// ---- DUTs/IO/Topology/Beckhoff_EK12xxEK1122_F8B8118B.TcDUT
{attribute 'GeneratedUsingTerminal: EK1122-0000-0018'}
{attribute addProperty BoxType "EK1122-0000-0018"}
{attribute addProperty Id "Beckhoff_EK12xxsub_EK1100EK1100_1FC0878B2A_0002_EK1200_7000_0000EK1200_013D0B490A_0001_EK1200_5000_0000EK1200_013D0B490"}
{attribute addProperty CRC "4172812683"}
{attribute addProperty Size "2"}
{attribute addProperty Name "Beckhoff EK12xxEK1122"}
TYPE Beckhoff_EK12xxEK1122_F8B8118B EXTENDS EK1122_1FC0878B :
STRUCT
	{attribute addProperty Name "Beckhoff EK12xxsub EK1100"}
	{attribute addProperty PreviousPort "Beckhoff EK12xxEK1122 : D"}
	Beckhoff_EK12xxsub_EK1100 : EK1100_1FC0878B;
	{attribute addProperty Name "A_0002(EK1200-7000-0000)"}
	{attribute addProperty PreviousPort "Beckhoff EK12xxsub EK1100 : C"}
	A_0002_EK1200_7000_0000 : EK1200_013D0B49;
	{attribute addProperty Name "A_0001(EK1200-5000-0000)"}
	{attribute addProperty PreviousPort "Beckhoff EK12xxsub EK1100 : C"}
	A_0001_EK1200_5000_0000 : EK1200_013D0B49;
END_STRUCT
END_TYPE

// ---- DUTs/IO/Topology/Beckhoff_EK12xx_F07DE953.TcDUT
{attribute 'GeneratedUsingTerminal: EK1100-0000-0018'}
{attribute addProperty BoxType "EK1100-0000-0018"}
{attribute addProperty Id "Beckhoff_EK12xxEK1122Beckhoff_EK12xxEK1122_F8B8118B2"}
{attribute addProperty CRC "4034783571"}
{attribute addProperty Size "2"}
{attribute addProperty Name "Beckhoff EK12xx"}
TYPE Beckhoff_EK12xx_F07DE953 EXTENDS EK1100_1FC0878B :
STRUCT
	{attribute addProperty Name "Beckhoff EK12xxEK1122"}
	{attribute addProperty PreviousPort "Beckhoff EK12xx : B"}
	Beckhoff_EK12xxEK1122 : Beckhoff_EK12xxEK1122_F8B8118B;
END_STRUCT
END_TYPE

// ---- DUTs/IO/Topology/Beckhoff_EK13xxEK1122_30D1B042.TcDUT
{attribute 'GeneratedUsingTerminal: EK1122-0000-0018'}
{attribute addProperty BoxType "EK1122-0000-0018"}
{attribute addProperty Id "Beckhoff_EK13xxsub_EK1100EK1100_1FC0878B2A_0001_EK1300_0000_0017EK1300_6BC01D146"}
{attribute addProperty CRC "819048514"}
{attribute addProperty Size "8"}
{attribute addProperty Name "Beckhoff EK13xxEK1122"}
TYPE Beckhoff_EK13xxEK1122_30D1B042 EXTENDS EK1122_1FC0878B :
STRUCT
	{attribute addProperty Name "Beckhoff EK13xxsub EK1100"}
	{attribute addProperty PreviousPort "Beckhoff EK13xxEK1122 : D"}
	Beckhoff_EK13xxsub_EK1100 : EK1100_1FC0878B;
	{attribute addProperty Name "A_0001(EK1300-0000-0017)"}
	{attribute addProperty PreviousPort "Beckhoff EK13xxsub EK1100 : C"}
	A_0001_EK1300_0000_0017 : EK1300_6BC01D14;
END_STRUCT
END_TYPE

// ---- DUTs/IO/Topology/Beckhoff_EK13xx_7663BCA8.TcDUT
{attribute 'GeneratedUsingTerminal: EK1100-0000-0018'}
{attribute addProperty BoxType "EK1100-0000-0018"}
{attribute addProperty Id "Beckhoff_EK13xxEK1122Beckhoff_EK13xxEK1122_30D1B0428A_0003_EK1322_0000_0017EK1322_6BC01D146A_0002_EK1310_0000_0017EK1310_6BC01D146"}
{attribute addProperty CRC "1986247848"}
{attribute addProperty Size "20"}
{attribute addProperty Name "Beckhoff EK13xx"}
TYPE Beckhoff_EK13xx_7663BCA8 EXTENDS EK1100_1FC0878B :
STRUCT
	{attribute addProperty Name "Beckhoff EK13xxEK1122"}
	{attribute addProperty PreviousPort "Beckhoff EK13xx : B"}
	Beckhoff_EK13xxEK1122 : Beckhoff_EK13xxEK1122_30D1B042;
	{attribute addProperty Name "A_0003(EK1322-0000-0017)"}
	{attribute addProperty PreviousPort "Beckhoff EK13xxEK1122 : C"}
	A_0003_EK1322_0000_0017 : EK1322_6BC01D14;
	{attribute addProperty Name "A_0002(EK1310-0000-0017)"}
	{attribute addProperty PreviousPort "A_0003(EK1322-0000-0017) : C"}
	A_0002_EK1310_0000_0017 : EK1310_6BC01D14;
END_STRUCT
END_TYPE

// ---- DUTs/IO/Topology/Beckhoff_EK15xxEK1122_1A424B62.TcDUT
{attribute 'GeneratedUsingTerminal: EK1122-0000-0018'}
{attribute addProperty BoxType "EK1122-0000-0018"}
{attribute addProperty Id "Beckhoff_EK15xxsub_EK1100EK1100_1FC0878B2A_0001_EK1501_0000_0016EK1501_957D888F6A_0002_EK1501_0000_0017EK1501_957D888F6A_0003_EK1501_0000_0018EK1501_957D888F6A_0004_EK1501_0000_0019EK1501_957D888F6A_0005_EK1501_0010_0016EK1501_957D888F6A_0006_EK1501_0010_0017EK1501_957D888F6A_0007_EK1501_0010_0018EK1501_957D888F6A_0008_EK1501_0100_0016EK1501_957D888F6A_0020_EK1541_0000_0016EK1541_957D888F6A_0021_EK1541_0000_0017EK1541_957D888F6A_0022_EK1541_0000_0018EK1541_957D888F6"}
{attribute addProperty CRC "440552290"}
{attribute addProperty Size "68"}
{attribute addProperty Name "Beckhoff EK15xxEK1122"}
TYPE Beckhoff_EK15xxEK1122_1A424B62 EXTENDS EK1122_1FC0878B :
STRUCT
	{attribute addProperty Name "Beckhoff EK15xxsub EK1100"}
	{attribute addProperty PreviousPort "Beckhoff EK15xxEK1122 : D"}
	Beckhoff_EK15xxsub_EK1100 : EK1100_1FC0878B;
	{attribute addProperty Name "A_0001(EK1501-0000-0016)"}
	{attribute addProperty PreviousPort "Beckhoff EK15xxsub EK1100 : C"}
	A_0001_EK1501_0000_0016 : EK1501_957D888F;
	{attribute addProperty Name "A_0002(EK1501-0000-0017)"}
	{attribute addProperty PreviousPort "A_0001(EK1501-0000-0016) : C"}
	A_0002_EK1501_0000_0017 : EK1501_957D888F;
	{attribute addProperty Name "A_0003(EK1501-0000-0018)"}
	{attribute addProperty PreviousPort "A_0002(EK1501-0000-0017) : C"}
	A_0003_EK1501_0000_0018 : EK1501_957D888F;
	{attribute addProperty Name "A_0004(EK1501-0000-0019)"}
	{attribute addProperty PreviousPort "A_0003(EK1501-0000-0018) : C"}
	A_0004_EK1501_0000_0019 : EK1501_957D888F;
	{attribute addProperty Name "A_0005(EK1501-0010-0016)"}
	{attribute addProperty PreviousPort "A_0004(EK1501-0000-0019) : C"}
	A_0005_EK1501_0010_0016 : EK1501_957D888F;
	{attribute addProperty Name "A_0006(EK1501-0010-0017)"}
	{attribute addProperty PreviousPort "A_0005(EK1501-0010-0016) : C"}
	A_0006_EK1501_0010_0017 : EK1501_957D888F;
	{attribute addProperty Name "A_0007(EK1501-0010-0018)"}
	{attribute addProperty PreviousPort "A_0006(EK1501-0010-0017) : C"}
	A_0007_EK1501_0010_0018 : EK1501_957D888F;
	{attribute addProperty Name "A_0008(EK1501-0100-0016)"}
	{attribute addProperty PreviousPort "A_0007(EK1501-0010-0018) : C"}
	A_0008_EK1501_0100_0016 : EK1501_957D888F;
	{attribute addProperty Name "A_0020(EK1541-0000-0016)"}
	{attribute addProperty PreviousPort "A_0008(EK1501-0100-0016) : C"}
	A_0020_EK1541_0000_0016 : EK1541_957D888F;
	{attribute addProperty Name "A_0021(EK1541-0000-0017)"}
	{attribute addProperty PreviousPort "A_0020(EK1541-0000-0016) : C"}
	A_0021_EK1541_0000_0017 : EK1541_957D888F;
	{attribute addProperty Name "A_0022(EK1541-0000-0018)"}
	{attribute addProperty PreviousPort "A_0021(EK1541-0000-0017) : C"}
	A_0022_EK1541_0000_0018 : EK1541_957D888F;
END_STRUCT
END_TYPE

// ---- DUTs/IO/Topology/Beckhoff_EK15xx_47CB6E2F.TcDUT
{attribute 'GeneratedUsingTerminal: EK1100-0000-0018'}
{attribute addProperty BoxType "EK1100-0000-0018"}
{attribute addProperty Id "Beckhoff_EK15xxEK1122Beckhoff_EK15xxEK1122_1A424B6268A_0025_EK1561_0000_0018EK1561_1FC0878B2A_0024_EK1561_0000_0017EK1561_1FC0878B2A_0023_EK1561_0000_0016EK1561_1FC0878B2A_0019_EK1521_0010_0020EK1521_1FC0878B2A_0018_EK1521_0010_0019EK1521_1FC0878B2A_0017_EK1521_0010_0018EK1521_1FC0878B2A_0016_EK1521_0010_0017EK1521_1FC0878B2A_0015_EK1521_0010_0016EK1521_1FC0878B2A_0014_EK1521_0000_0021EK1521_1FC0878B2A_0013_EK1521_0000_0020EK1521_1FC0878B2A_0012_EK1521_0000_0019EK1521_1FC0878B2A_0011_EK1521_0000_0018EK1521_1FC0878B2A_0010_EK1521_0000_0017EK1521_1FC0878B2A_0009_EK1521_0000_0016EK1521_1FC0878B2"}
{attribute addProperty CRC "1204514351"}
{attribute addProperty Size "96"}
{attribute addProperty Name "Beckhoff EK15xx"}
TYPE Beckhoff_EK15xx_47CB6E2F EXTENDS EK1100_1FC0878B :
STRUCT
	{attribute addProperty Name "Beckhoff EK15xxEK1122"}
	{attribute addProperty PreviousPort "Beckhoff EK15xx : B"}
	Beckhoff_EK15xxEK1122 : Beckhoff_EK15xxEK1122_1A424B62;
	{attribute addProperty Name "A_0025(EK1561-0000-0018)"}
	{attribute addProperty PreviousPort "Beckhoff EK15xxEK1122 : C"}
	A_0025_EK1561_0000_0018 : EK1561_1FC0878B;
	{attribute addProperty Name "A_0024(EK1561-0000-0017)"}
	{attribute addProperty PreviousPort "A_0025(EK1561-0000-0018) : C"}
	A_0024_EK1561_0000_0017 : EK1561_1FC0878B;
	{attribute addProperty Name "A_0023(EK1561-0000-0016)"}
	{attribute addProperty PreviousPort "A_0024(EK1561-0000-0017) : C"}
	A_0023_EK1561_0000_0016 : EK1561_1FC0878B;
	{attribute addProperty Name "A_0019(EK1521-0010-0020)"}
	{attribute addProperty PreviousPort "A_0023(EK1561-0000-0016) : C"}
	A_0019_EK1521_0010_0020 : EK1521_1FC0878B;
	{attribute addProperty Name "A_0018(EK1521-0010-0019)"}
	{attribute addProperty PreviousPort "A_0019(EK1521-0010-0020) : C"}
	A_0018_EK1521_0010_0019 : EK1521_1FC0878B;
	{attribute addProperty Name "A_0017(EK1521-0010-0018)"}
	{attribute addProperty PreviousPort "A_0018(EK1521-0010-0019) : C"}
	A_0017_EK1521_0010_0018 : EK1521_1FC0878B;
	{attribute addProperty Name "A_0016(EK1521-0010-0017)"}
	{attribute addProperty PreviousPort "A_0017(EK1521-0010-0018) : C"}
	A_0016_EK1521_0010_0017 : EK1521_1FC0878B;
	{attribute addProperty Name "A_0015(EK1521-0010-0016)"}
	{attribute addProperty PreviousPort "A_0016(EK1521-0010-0017) : C"}
	A_0015_EK1521_0010_0016 : EK1521_1FC0878B;
	{attribute addProperty Name "A_0014(EK1521-0000-0021)"}
	{attribute addProperty PreviousPort "A_0015(EK1521-0010-0016) : C"}
	A_0014_EK1521_0000_0021 : EK1521_1FC0878B;
	{attribute addProperty Name "A_0013(EK1521-0000-0020)"}
	{attribute addProperty PreviousPort "A_0014(EK1521-0000-0021) : C"}
	A_0013_EK1521_0000_0020 : EK1521_1FC0878B;
	{attribute addProperty Name "A_0012(EK1521-0000-0019)"}
	{attribute addProperty PreviousPort "A_0013(EK1521-0000-0020) : C"}
	A_0012_EK1521_0000_0019 : EK1521_1FC0878B;
	{attribute addProperty Name "A_0011(EK1521-0000-0018)"}
	{attribute addProperty PreviousPort "A_0012(EK1521-0000-0019) : C"}
	A_0011_EK1521_0000_0018 : EK1521_1FC0878B;
	{attribute addProperty Name "A_0010(EK1521-0000-0017)"}
	{attribute addProperty PreviousPort "A_0011(EK1521-0000-0018) : C"}
	A_0010_EK1521_0000_0017 : EK1521_1FC0878B;
	{attribute addProperty Name "A_0009(EK1521-0000-0016)"}
	{attribute addProperty PreviousPort "A_0010(EK1521-0000-0017) : C"}
	A_0009_EK1521_0000_0016 : EK1521_1FC0878B;
END_STRUCT
END_TYPE

// ---- DUTs/IO/Topology/Beckhoff_EK18xxEK1122_F7FACD4D.TcDUT
{attribute 'GeneratedUsingTerminal: EK1122-0000-0018'}
{attribute addProperty BoxType "EK1122-0000-0018"}
{attribute addProperty Id "Beckhoff_EK18xxsub_EK1100EK1100_1FC0878B2A_0001_EK1814_0000_0016EK1814_F6D9A8D112A_0002_EK1814_0000_0017EK1814_F6D9A8D112A_0003_EK1814_0000_0018EK1814_F6D9A8D112A_0004_EK1814_0000_0019EK1814_F6D9A8D112A_0005_EK1818_0000_0016EK1818_6B19C24E16A_0006_EK1818_0000_0017EK1818_6B19C24E16A_0007_EK1818_0000_0018EK1818_6B19C24E16A_0008_EK1828_0000_0016EK1828_56D6F88716A_0009_EK1828_0000_0017EK1828_56D6F88716A_0010_EK1828_0000_0018EK1828_56D6F88716A_0011_EK1828_0010_0016EK1828_E2806B9511A_0012_EK1828_0010_0017EK1828_E2806B9511A_0013_EK1828_0010_0018EK1828_E2806B9511"}
{attribute addProperty CRC "4160408909"}
{attribute addProperty Size "179"}
{attribute addProperty Name "Beckhoff EK18xxEK1122"}
TYPE Beckhoff_EK18xxEK1122_F7FACD4D EXTENDS EK1122_1FC0878B :
STRUCT
	{attribute addProperty Name "Beckhoff EK18xxsub EK1100"}
	{attribute addProperty PreviousPort "Beckhoff EK18xxEK1122 : D"}
	Beckhoff_EK18xxsub_EK1100 : EK1100_1FC0878B;
	{attribute addProperty Name "A_0001(EK1814-0000-0016)"}
	{attribute addProperty PreviousPort "Beckhoff EK18xxsub EK1100 : C"}
	A_0001_EK1814_0000_0016 : EK1814_F6D9A8D1;
	{attribute addProperty Name "A_0002(EK1814-0000-0017)"}
	{attribute addProperty PreviousPort "A_0001(EK1814-0000-0016) : C"}
	A_0002_EK1814_0000_0017 : EK1814_F6D9A8D1;
	{attribute addProperty Name "A_0003(EK1814-0000-0018)"}
	{attribute addProperty PreviousPort "A_0002(EK1814-0000-0017) : C"}
	A_0003_EK1814_0000_0018 : EK1814_F6D9A8D1;
	{attribute addProperty Name "A_0004(EK1814-0000-0019)"}
	{attribute addProperty PreviousPort "A_0003(EK1814-0000-0018) : C"}
	A_0004_EK1814_0000_0019 : EK1814_F6D9A8D1;
	{attribute addProperty Name "A_0005(EK1818-0000-0016)"}
	{attribute addProperty PreviousPort "A_0004(EK1814-0000-0019) : C"}
	A_0005_EK1818_0000_0016 : EK1818_6B19C24E;
	{attribute addProperty Name "A_0006(EK1818-0000-0017)"}
	{attribute addProperty PreviousPort "A_0005(EK1818-0000-0016) : C"}
	A_0006_EK1818_0000_0017 : EK1818_6B19C24E;
	{attribute addProperty Name "A_0007(EK1818-0000-0018)"}
	{attribute addProperty PreviousPort "A_0006(EK1818-0000-0017) : C"}
	A_0007_EK1818_0000_0018 : EK1818_6B19C24E;
	{attribute addProperty Name "A_0008(EK1828-0000-0016)"}
	{attribute addProperty PreviousPort "A_0007(EK1818-0000-0018) : C"}
	A_0008_EK1828_0000_0016 : EK1828_56D6F887;
	{attribute addProperty Name "A_0009(EK1828-0000-0017)"}
	{attribute addProperty PreviousPort "A_0008(EK1828-0000-0016) : C"}
	A_0009_EK1828_0000_0017 : EK1828_56D6F887;
	{attribute addProperty Name "A_0010(EK1828-0000-0018)"}
	{attribute addProperty PreviousPort "A_0009(EK1828-0000-0017) : C"}
	A_0010_EK1828_0000_0018 : EK1828_56D6F887;
	{attribute addProperty Name "A_0011(EK1828-0010-0016)"}
	{attribute addProperty PreviousPort "A_0010(EK1828-0000-0018) : C"}
	A_0011_EK1828_0010_0016 : EK1828_E2806B95;
	{attribute addProperty Name "A_0012(EK1828-0010-0017)"}
	{attribute addProperty PreviousPort "A_0011(EK1828-0010-0016) : C"}
	A_0012_EK1828_0010_0017 : EK1828_E2806B95;
	{attribute addProperty Name "A_0013(EK1828-0010-0018)"}
	{attribute addProperty PreviousPort "A_0012(EK1828-0010-0017) : C"}
	A_0013_EK1828_0010_0018 : EK1828_E2806B95;
END_STRUCT
END_TYPE

// ---- DUTs/IO/Topology/Beckhoff_EK18xx_88ED272B.TcDUT
{attribute 'GeneratedUsingTerminal: EK1100-0000-0018'}
{attribute addProperty BoxType "EK1100-0000-0018"}
{attribute addProperty Id "Beckhoff_EK18xxEK1122Beckhoff_EK18xxEK1122_F7FACD4D179"}
{attribute addProperty CRC "2297243435"}
{attribute addProperty Size "179"}
{attribute addProperty Name "Beckhoff EK18xx"}
TYPE Beckhoff_EK18xx_88ED272B EXTENDS EK1100_1FC0878B :
STRUCT
	{attribute addProperty Name "Beckhoff EK18xxEK1122"}
	{attribute addProperty PreviousPort "Beckhoff EK18xx : B"}
	Beckhoff_EK18xxEK1122 : Beckhoff_EK18xxEK1122_F7FACD4D;
END_STRUCT
END_TYPE

// ---- DUTs/IO/Topology/Beckhoff_EKM1xxxEK1122_F03648A5.TcDUT
{attribute 'GeneratedUsingTerminal: EK1122-0000-0018'}
{attribute addProperty BoxType "EK1122-0000-0018"}
{attribute addProperty Id "Beckhoff_EKM1xxxsub_EK1100EK1100_1FC0878B2A_0001_EKM1101_0000_0016EKM1101_7F41762282A_0002_EKM1101_0000_0017EKM1101_7F41762282A_0003_EKM1101_0000_0018EKM1101_7F41762282A_0004_EKM1101_0000_0019EKM1101_7F41762282A_0005_EKM1101_0000_0020EKM1101_7F41762282"}
{attribute addProperty CRC "4030089381"}
{attribute addProperty Size "412"}
{attribute addProperty Name "Beckhoff EKM1xxxEK1122"}
TYPE Beckhoff_EKM1xxxEK1122_F03648A5 EXTENDS EK1122_1FC0878B :
STRUCT
	{attribute addProperty Name "Beckhoff EKM1xxxsub EK1100"}
	{attribute addProperty PreviousPort "Beckhoff EKM1xxxEK1122 : D"}
	Beckhoff_EKM1xxxsub_EK1100 : EK1100_1FC0878B;
	{attribute addProperty Name "A_0001(EKM1101-0000-0016)"}
	{attribute addProperty PreviousPort "Beckhoff EKM1xxxsub EK1100 : C"}
	A_0001_EKM1101_0000_0016 : EKM1101_7F417622;
	{attribute addProperty Name "A_0002(EKM1101-0000-0017)"}
	{attribute addProperty PreviousPort "A_0001(EKM1101-0000-0016) : C"}
	A_0002_EKM1101_0000_0017 : EKM1101_7F417622;
	{attribute addProperty Name "A_0003(EKM1101-0000-0018)"}
	{attribute addProperty PreviousPort "A_0002(EKM1101-0000-0017) : C"}
	A_0003_EKM1101_0000_0018 : EKM1101_7F417622;
	{attribute addProperty Name "A_0004(EKM1101-0000-0019)"}
	{attribute addProperty PreviousPort "A_0003(EKM1101-0000-0018) : C"}
	A_0004_EKM1101_0000_0019 : EKM1101_7F417622;
	{attribute addProperty Name "A_0005(EKM1101-0000-0020)"}
	{attribute addProperty PreviousPort "A_0004(EKM1101-0000-0019) : C"}
	A_0005_EKM1101_0000_0020 : EKM1101_7F417622;
END_STRUCT
END_TYPE

// ---- DUTs/IO/Topology/Beckhoff_EKM1xxx_245084ED.TcDUT
{attribute 'GeneratedUsingTerminal: EK1100-0000-0018'}
{attribute addProperty BoxType "EK1100-0000-0018"}
{attribute addProperty Id "Beckhoff_EKM1xxxEK1122Beckhoff_EKM1xxxEK1122_F03648A5412"}
{attribute addProperty CRC "609256685"}
{attribute addProperty Size "412"}
{attribute addProperty Name "Beckhoff EKM1xxx"}
TYPE Beckhoff_EKM1xxx_245084ED EXTENDS EK1100_1FC0878B :
STRUCT
	{attribute addProperty Name "Beckhoff EKM1xxxEK1122"}
	{attribute addProperty PreviousPort "Beckhoff EKM1xxx : B"}
	Beckhoff_EKM1xxxEK1122 : Beckhoff_EKM1xxxEK1122_F03648A5;
END_STRUCT
END_TYPE

// ---- DUTs/IO/Topology/Beckhoff_EKx9xxEK1122_41BF98AA.TcDUT
{attribute 'GeneratedUsingTerminal: EK1122-0000-0018'}
{attribute addProperty BoxType "EK1122-0000-0018"}
{attribute addProperty Id "Beckhoff_EKx9xxsub_EK1100EK1100_1FC0878B2A_0001_EK1960_0000_0019EK1960_14394C51142A_0002_EK1960_0000_0021EK1960_9900B192138A_0003_EK1960_0008_0019EK1960_14394C51142A_0004_EK1960_0008_0021EK1960_9900B192138A_0005_EK1960_2600_0019EK1960_BAE25DEC148A_0006_EK1960_2600_0021EK1960_2415CDAE148A_0007_EK1960_2608_0019EK1960_BAE25DEC148A_0008_EK1960_2608_0021EK1960_2415CDAE148"}
{attribute addProperty CRC "1103075498"}
{attribute addProperty Size "1154"}
{attribute addProperty Name "Beckhoff EKx9xxEK1122"}
TYPE Beckhoff_EKx9xxEK1122_41BF98AA EXTENDS EK1122_1FC0878B :
STRUCT
	{attribute addProperty Name "Beckhoff EKx9xxsub EK1100"}
	{attribute addProperty PreviousPort "Beckhoff EKx9xxEK1122 : D"}
	Beckhoff_EKx9xxsub_EK1100 : EK1100_1FC0878B;
	{attribute addProperty Name "A_0001(EK1960-0000-0019)"}
	{attribute addProperty PreviousPort "Beckhoff EKx9xxsub EK1100 : C"}
	A_0001_EK1960_0000_0019 : EK1960_14394C51;
	{attribute addProperty Name "A_0002(EK1960-0000-0021)"}
	{attribute addProperty PreviousPort "A_0001(EK1960-0000-0019) : C"}
	A_0002_EK1960_0000_0021 : EK1960_9900B192;
	{attribute addProperty Name "A_0003(EK1960-0008-0019)"}
	{attribute addProperty PreviousPort "A_0002(EK1960-0000-0021) : C"}
	A_0003_EK1960_0008_0019 : EK1960_14394C51;
	{attribute addProperty Name "A_0004(EK1960-0008-0021)"}
	{attribute addProperty PreviousPort "A_0003(EK1960-0008-0019) : C"}
	A_0004_EK1960_0008_0021 : EK1960_9900B192;
	{attribute addProperty Name "A_0005(EK1960-2600-0019)"}
	{attribute addProperty PreviousPort "A_0004(EK1960-0008-0021) : C"}
	A_0005_EK1960_2600_0019 : EK1960_BAE25DEC;
	{attribute addProperty Name "A_0006(EK1960-2600-0021)"}
	{attribute addProperty PreviousPort "A_0005(EK1960-2600-0019) : C"}
	A_0006_EK1960_2600_0021 : EK1960_2415CDAE;
	{attribute addProperty Name "A_0007(EK1960-2608-0019)"}
	{attribute addProperty PreviousPort "A_0006(EK1960-2600-0021) : C"}
	A_0007_EK1960_2608_0019 : EK1960_BAE25DEC;
	{attribute addProperty Name "A_0008(EK1960-2608-0021)"}
	{attribute addProperty PreviousPort "A_0007(EK1960-2608-0019) : C"}
	A_0008_EK1960_2608_0021 : EK1960_2415CDAE;
END_STRUCT
END_TYPE

// ---- DUTs/IO/Topology/Beckhoff_EKx9xx_36A98EAE.TcDUT
{attribute 'GeneratedUsingTerminal: EK1100-0000-0018'}
{attribute addProperty BoxType "EK1100-0000-0018"}
{attribute addProperty Id "Beckhoff_EKx9xxEK1122Beckhoff_EKx9xxEK1122_41BF98AA1154"}
{attribute addProperty CRC "917081774"}
{attribute addProperty Size "1154"}
{attribute addProperty Name "Beckhoff EKx9xx"}
TYPE Beckhoff_EKx9xx_36A98EAE EXTENDS EK1100_1FC0878B :
STRUCT
	{attribute addProperty Name "Beckhoff EKx9xxEK1122"}
	{attribute addProperty PreviousPort "Beckhoff EKx9xx : B"}
	Beckhoff_EKx9xxEK1122 : Beckhoff_EKx9xxEK1122_41BF98AA;
END_STRUCT
END_TYPE

// ---- DUTs/IO/Topology/Beckhoff_EKxxxx_0080EK1122_9CBA35F2.TcDUT
{attribute 'GeneratedUsingTerminal: EK1122-0000-0018'}
{attribute addProperty BoxType "EK1122-0000-0018"}
{attribute addProperty Id "Beckhoff_EKxxxx_0080sub_EK1100EK1100_1FC0878B2"}
{attribute addProperty CRC "2629449202"}
{attribute addProperty Size "2"}
{attribute addProperty Name "Beckhoff EKxxxx-0080EK1122"}
TYPE Beckhoff_EKxxxx_0080EK1122_9CBA35F2 EXTENDS EK1122_1FC0878B :
STRUCT
	{attribute addProperty Name "Beckhoff EKxxxx-0080sub EK1100"}
	{attribute addProperty PreviousPort "Beckhoff EKxxxx-0080EK1122 : D"}
	Beckhoff_EKxxxx_0080sub_EK1100 : EK1100_1FC0878B;
END_STRUCT
END_TYPE

// ---- DUTs/IO/Topology/Beckhoff_EKxxxx_0080_9DDEF925.TcDUT
{attribute 'GeneratedUsingTerminal: EK1100-0000-0018'}
{attribute addProperty BoxType "EK1100-0000-0018"}
{attribute addProperty Id "Beckhoff_EKxxxx_0080EK1122Beckhoff_EKxxxx_0080EK1122_9CBA35F22A_0006_EK1122_0080_0019EK1122_1FC0878B2A_0005_EK1122_0080_0018EK1122_1FC0878B2A_0004_EK1122_0080_0017EK1122_1FC0878B2"}
{attribute addProperty CRC "2648635685"}
{attribute addProperty Size "8"}
{attribute addProperty Name "Beckhoff EKxxxx-0080"}
TYPE Beckhoff_EKxxxx_0080_9DDEF925 EXTENDS EK1100_1FC0878B :
STRUCT
	{attribute addProperty Name "Beckhoff EKxxxx-0080EK1122"}
	{attribute addProperty PreviousPort "Beckhoff EKxxxx-0080 : B"}
	Beckhoff_EKxxxx_0080EK1122 : Beckhoff_EKxxxx_0080EK1122_9CBA35F2;
	{attribute addProperty Name "A_0006(EK1122-0080-0019)"}
	{attribute addProperty PreviousPort "Beckhoff EKxxxx-0080EK1122 : C"}
	A_0006_EK1122_0080_0019 : EK1122_1FC0878B;
	{attribute addProperty Name "A_0005(EK1122-0080-0018)"}
	{attribute addProperty PreviousPort "A_0006(EK1122-0080-0019) : C"}
	A_0005_EK1122_0080_0018 : EK1122_1FC0878B;
	{attribute addProperty Name "A_0004(EK1122-0080-0017)"}
	{attribute addProperty PreviousPort "A_0005(EK1122-0080-0018) : C"}
	A_0004_EK1122_0080_0017 : EK1122_1FC0878B;
END_STRUCT
END_TYPE

// ---- DUTs/IO/Topology/EtherCAT_Master_EKxxxx_2095F716.TcDUT
{attribute 'GeneratedUsingTerminal: IODEVICETYPE_ETHERCATPROT'}
{attribute addProperty BoxType "IODEVICETYPE_ETHERCATPROT"}
{attribute addProperty Id "Beckhoff_EK11xxBeckhoff_EK11xx_811529C670Beckhoff_EK12xxBeckhoff_EK12xx_F07DE9532Beckhoff_EK13xxBeckhoff_EK13xx_7663BCA820Beckhoff_EK15xxBeckhoff_EK15xx_47CB6E2F96Beckhoff_EK18xxBeckhoff_EK18xx_88ED272B179Beckhoff_EKM1xxxBeckhoff_EKM1xxx_245084ED412Beckhoff_EKx9xxBeckhoff_EKx9xx_36A98EAE1154Beckhoff_EKxxxx_0080Beckhoff_EKxxxx_0080_9DDEF9258SyncUnitsSyncUnits_99E584AF18InputsInputs_25A0042B160OutputsOutputs_2397A10E106InfoDataInfoData_E68C61CD28"}
{attribute addProperty CRC "546699030"}
{attribute addProperty Size "2253"}
{attribute addProperty Name "EtherCAT Master EKxxxx"}
TYPE EtherCAT_Master_EKxxxx_2095F716 EXTENDS EtcMasterBase_62654B43 :
STRUCT
	{attribute addProperty Name "Beckhoff EK11xx"}
	{attribute addProperty PreviousPort "EtherCAT Master EKxxxx : Master"}
	Beckhoff_EK11xx : Beckhoff_EK11xx_811529C6;
	{attribute addProperty Name "Beckhoff EK12xx"}
	{attribute addProperty PreviousPort "A_0014(EK1110-0000-0000) : B"}
	Beckhoff_EK12xx : Beckhoff_EK12xx_F07DE953;
	{attribute addProperty Name "Beckhoff EK13xx"}
	{attribute addProperty PreviousPort "Beckhoff EK12xx : C"}
	Beckhoff_EK13xx : Beckhoff_EK13xx_7663BCA8;
	{attribute addProperty Name "Beckhoff EK15xx"}
	{attribute addProperty PreviousPort "A_0002(EK1310-0000-0017) : B"}
	Beckhoff_EK15xx : Beckhoff_EK15xx_47CB6E2F;
	{attribute addProperty Name "Beckhoff EK18xx"}
	{attribute addProperty PreviousPort "Beckhoff EK15xx : C"}
	Beckhoff_EK18xx : Beckhoff_EK18xx_88ED272B;
	{attribute addProperty Name "Beckhoff EKM1xxx"}
	{attribute addProperty PreviousPort "Beckhoff EK18xx : C"}
	Beckhoff_EKM1xxx : Beckhoff_EKM1xxx_245084ED;
	{attribute addProperty Name "Beckhoff EKx9xx"}
	{attribute addProperty PreviousPort "Beckhoff EKM1xxx : C"}
	Beckhoff_EKx9xx : Beckhoff_EKx9xx_36A98EAE;
	{attribute addProperty Name "Beckhoff EKxxxx-0080"}
	{attribute addProperty PreviousPort "Beckhoff EKx9xx : C"}
	Beckhoff_EKxxxx_0080 : Beckhoff_EKxxxx_0080_9DDEF925;
	{attribute addProperty Name "SyncUnits"}
	SyncUnits : SyncUnits_99E584AF;
	{attribute addProperty Name "Inputs"}
	Inputs : Inputs_25A0042B;
	{attribute addProperty Name "Outputs"}
	Outputs : Outputs_2397A10E;
	{attribute addProperty Name "InfoData"}
	InfoData : InfoData_E68C61CD;
END_STRUCT
END_TYPE

// ---- DUTs/IO/Base/EtcSlaveBase_82538BE2.TcDUT

TYPE EtcSlaveBase_82538BE2 :
STRUCT
END_STRUCT
END_TYPE

// ---- DUTs/IO/Base/EtcSlaveBase_82538BE2.TcDUT

TYPE EtcSlaveBase_82538BE2 :
STRUCT
END_STRUCT
END_TYPE

// ---- DUTs/IO/Base/EtcSlaveBase_82538BE2.TcDUT

TYPE EtcSlaveBase_82538BE2 :
STRUCT
END_STRUCT
END_TYPE

// ---- DUTs/IO/Base/EtcSlaveTerminalBase_947E5A46.TcDUT

{attribute clr[Container(Layout.Stack)]}
{attribute clr[Group(Layout.GroupBox)]}
{attribute addProperty PreviousPort "Unknown"}
TYPE EtcSlaveTerminalBase_947E5A46 EXTENDS EtcSlaveBase_82538BE2 :
STRUCT
END_STRUCT
END_TYPE

// ---- DUTs/IO/Base/EtcSlaveBoxBase_77A0E4A7.TcDUT

{attribute clr[Container(Layout.Stack)]}
{attribute clr[Group(Layout.GroupBox)]}
{attribute addProperty PreviousPort "Unknown"}
TYPE EtcSlaveBoxBase_77A0E4A7 EXTENDS EtcSlaveBase_82538BE2 :
STRUCT
END_STRUCT
END_TYPE

// ---- DUTs/IO/Base/EtcSlaveEndTerminalBase_866C7F0C.TcDUT

{attribute clr[Container(Layout.Stack)]}
{attribute clr[Group(Layout.GroupBox)]}
{attribute addProperty PreviousPort "Unknown"}
TYPE EtcSlaveEndTerminalBase_866C7F0C EXTENDS EtcSlaveBase_82538BE2 :
STRUCT
END_STRUCT
END_TYPE

// ---- DUTs/IO/Base/InputBase_8311D824.TcDUT

TYPE InputBase_8311D824 :
STRUCT
END_STRUCT
END_TYPE

// ---- DUTs/IO/Base/OutputBase_10CEE7DE.TcDUT

TYPE OutputBase_10CEE7DE :
STRUCT
END_STRUCT
END_TYPE

// ---- DUTs/IO/Base/EtcMasterBase_62654B43.TcDUT

TYPE EtcMasterBase_62654B43 :
STRUCT
END_STRUCT
END_TYPE

// ---- GVLs/GVL_iXlinker.TcGVL
{attribute 'qualified_only'}
VAR_GLOBAL
		EtherCAT_Master_EKxxxx : EtherCAT_Master_EKxxxx_2095F716;
END_VAR

// ---- POUs/MAIN.TcPOU
PROGRAM MAIN
VAR
END_VAR

END_PROGRAM
